FUNCTION_BLOCK MultiTrigger
VAR
	Output AT %Q*: BOOL;
	Start: BOOL := FALSE;
	Active: BOOL := FALSE;
	TicksHigh: UINT := 100;
	TicksLow: UINT := 100;
	NumTrigger: INT := 20;
	NumCurrent: INT := 0;
	TickCount: UINT := 0;
	Stop: BOOL := FALSE;
END_VAR

TicksHigh := MAX(1, TicksHigh);
TicksLow := MAX(1, TicksLow);

IF Start THEN
	Active := TRUE;
	Start := FALSE;
	NumCurrent := 0;
END_IF

IF Stop THEN
	Active := FALSE;
	Output := FALSE;
	Stop := FALSE;
END_IF

IF Active THEN
	TickCount := TickCount + 1;
	IF Output THEN
		IF TickCount >= TicksHigh THEN
			Output := FALSE;
			TickCount := 0;
			IF NumCurrent = NumTrigger THEN
				Active := FALSE;
			END_IF
		END_IF
	ELSE
		IF TickCount >= TicksLow THEN
			NumCurrent := NumCurrent + 1;
			Output := TRUE;
			TickCount := 0;
		END_IF
	END_IF
END_IF

END_FUNCTION_BLOCK

(* stored: Version 1.1.0.1, ProductVersion 3.1.4024.15
   POU MultiTrigger: Id {5036bf31-ff01-4751-b839-f1812de29666}, SpecialFunc None *)
